// TIA Portal V20 export
VAR_GLOBAL   // PLC tag table "LGR_Const_StopClass"
END_VAR
VAR_GLOBAL CONSTANT   // user constants
   STOP_NORMAL : USInt := 0;
   STOP_FAST : USInt := 1;
END_VAR
